ABB RobotStudio station: LearningSolution_20201010-132329.rsstn

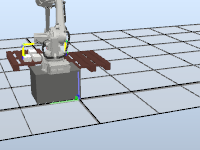
Station LearningSolution (saved by RobotStudio 20.2.9116.0)
Controller LearningController1, task T_ROB1: task frame (RAPID world) sits at (316.67, 323.87, 500) mm in the station
Controller LearningController1
  mechanical unit ROB_1: IRB4600_20_250_C_01, 6 joints, base frame (0, 0, 0) mm
Layout (positions relative to the parent item):
  - IRB4600_20_250_C_01 [mechanism, from Robots\IRB4600_20_250_C_G_01.rslib] at (316.67, 323.87, 500) mm; joint values [-0.1763, 1.0283, -0.0561, 0, 0.5986, 2.9653] (rad or m)
  - Table [part] at (1374.27, -5589.12, 0) mm
  - Engine Block [part] at (1630.97, -5278.43, 365.71) mm, rotated rx 90.36 ry 0 rz 0 deg
  - Base [part] at (57.41, 707.37, 0) mm, rotated rx 90 ry 0 rz 0 deg
  - Euro Pallet from [graphiccomponentgroup, from Equipment\Euro Pallet.rslib] at (1956.13, 0, 0) mm
    - Body 1 [part, from Equipment\Euro Pallet.rslib]
  - Box [part] at (2148.53, 78.03, 244.24) mm, rotated rx -90 ry 0 rz 0 deg
  - Box_2 [part] at (2173.15, 266.46, 244.24) mm, rotated rx -90 ry 0 rz 0 deg
  - Box_3 [part] at (2215.66, 466.33, 244.24) mm, rotated rx -90 ry 0 rz 0 deg
  - Box_4 [part] at (2622.54, 269.44, 244.24) mm, rotated rx -90 ry 0 rz 0 deg
  - Euro Pallet to [graphiccomponentgroup, from Equipment\Euro Pallet.rslib] at (1348.12, -1157.59, 0) mm
    - Body 1 [part, from Equipment\Euro Pallet.rslib]
  - Frame_2 [frame] at (-21.5, 24, 57.4) mm
Collision set CollisionSet_1: Box, Box_2, Box_3, Box_4 against , near miss 0 m
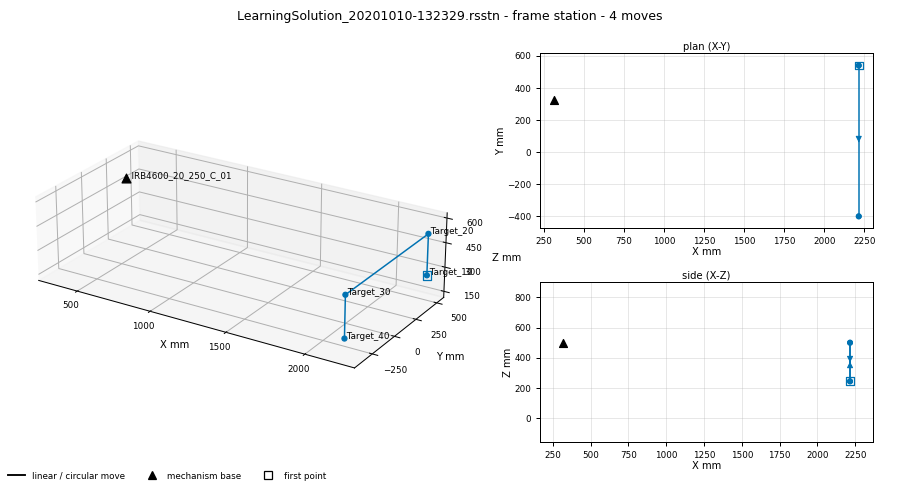
[picture p0: tool path of LearningSolution_20201010-132329.rsstn in frame station, 4 of 4 moves have a stored position in this frame; points joined in program order, loops and branches not executed]
Targets, tools, work objects and paths stored in the station, written as RAPID:
! task T_ROB1
MODULE CalibData
  PERS tooldata MyTool:=[TRUE,[[31.792631019,0,229.638935148],[0.945518576,0,0.325568154,0]],[1,[0,0,1],[1,0,0,0],0,0,0]];
ENDMODULE

! task T_ROB1
MODULE Module1
  CONST robtarget Target_10:=[[1898.989,216.715052945,-255.022709531],[0,1,0,0],[0,0,0,0],[9E+09,9E+09,9E+09,9E+09,9E+09,9E+09]];
  CONST robtarget Target_20:=[[1898.989,216.715052945,0.000290469],[0,1,0,0],[0,0,0,0],[9E+09,9E+09,9E+09,9E+09,9E+09,9E+09]];
  CONST robtarget Target_30:=[[1898.989,-723.871947055,0.000290469],[0,1,0,0],[0,0,0,0],[9E+09,9E+09,9E+09,9E+09,9E+09,9E+09]];
  CONST robtarget Target_40:=[[1898.989,-723.871947055,-256.499709531],[0,1,0,0],[0,0,0,0],[9E+09,9E+09,9E+09,9E+09,9E+09,9E+09]];
  PROC main()
  ENDPROC
  PROC Path_10()
    MoveL Target_10,v600,z5,tool0\WObj:=wobj0;
    MoveL Target_20,v600,z5,tool0\WObj:=wobj0;
    MoveL Target_30,v600,z5,tool0\WObj:=wobj0;
    MoveL Target_40,v600,z5,tool0\WObj:=wobj0;
  ENDPROC
ENDMODULE

